INTERFACE I_BrakeShareData

PROPERTY AxisState : MC_AxisStates
GET
END_GET
END_PROPERTY

END_INTERFACE

(* stored: Version 1.1.0.1
   Itf I_BrakeShareData: Id {14c61b0f-df7f-4928-9d16-c71acb1efb28}
   Property AxisState: Id {ba097a17-7813-4cd5-8d3b-6799b9ffbe35}
   Get Get: Id {a2b9a892-bb8b-475b-bda0-a7d3aa1d87df} *)
